(* Logix 5000 project; controller AMANA_DC_PLANT_01 vendor 1 type 14 code 164 rev 31.12; software revision 31.02; part 3 of 9 *)
(* tags used below, declared in another part *)
   Break1_Hour : DINT;
   Break1_Hour_String : STRING_4;
   Break1_Length : DINT;
   Break1_Min : DINT;
   Break1_Min_String : STRING_4;
   Break2_Hour : DINT;
   Break2_Hour_String : STRING_4;
   Break2_Length : DINT;
   Break2_Min : DINT;
   Break2_Min_String : STRING_4;
   End_Hour : DINT;
   End_Hour_String : STRING_4;
   End_Min : DINT;
   End_Min_String : STRING_4;
   Lunch_Hour : DINT;
   Lunch_Hour_String : STRING_4;
   Lunch_Length : DINT;
   Lunch_Min : DINT;
   Lunch_Min_String : STRING_4;
   PreviousCount : DINT;
   Shift_Reset : BOOL;
   Start_Hour : DINT;
   Start_Hour_String : STRING_4;
   Start_Min : DINT;
   Start_Min_String : STRING_4;
   theoreticalUnitsReal : REAL;
   ay : REAL;
   fifi_unload : DINT;
   LN00_Schedule : UDT_Current_Status;
   LN00_ScheduleUnits_Produced_from_line : DINT;
   LN00_to_DC1_Main_Messages_0 : DINT[40];
   LN00_Toggle_CountSource : BOOL;
   LN00_Weekly_Schedule : UDT_Weekly_Schedule;
   null : STRING;
   Previous_Shift_Count : DINT;
   scc : CONTROL;   // Shift Count History
   Shift_count_history : DINT[62];
   Shift_reset_timer : TIMER;
   THEORETICAL_TEST : BOOL;
(* LN00, continued *)

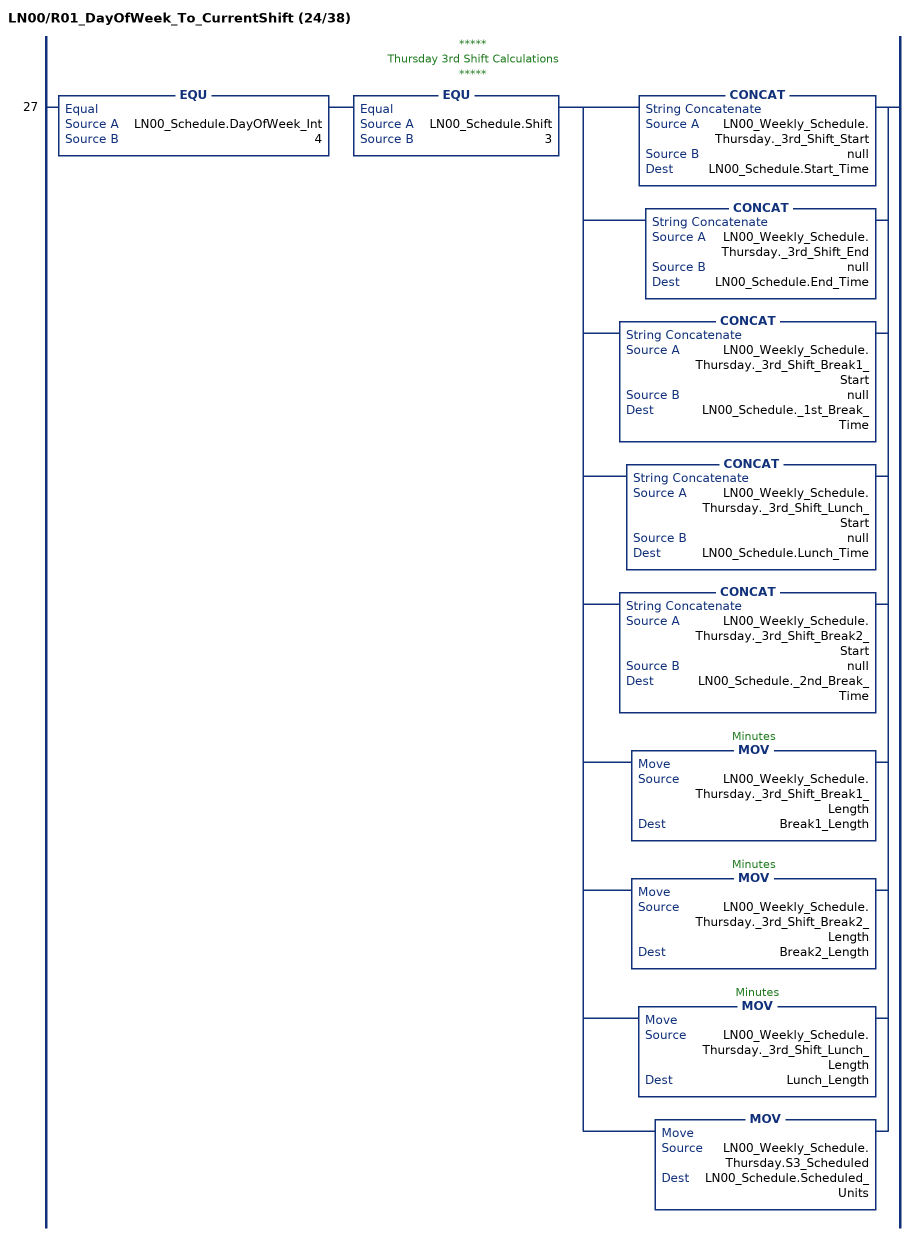
   [picture p24: LN00/R01_DayOfWeek_To_CurrentShift rungs 27-27]
   // *****
   // Thursday 3rd Shift Calculations
   // *****
   27: EQU(LN00_Schedule.DayOfWeek_Int,4)EQU(LN00_Schedule.Shift,3)[CONCAT(LN00_Weekly_Schedule.Thursday._3rd_Shift_Start,null,LN00_Schedule.Start_Time) ,CONCAT(LN00_Weekly_Schedule.Thursday._3rd_Shift_End,null,LN00_Schedule.End_Time) ,CONCAT(LN00_Weekly_Schedule.Thursday._3rd_Shift_Break1_Start,null,LN00_Schedule._1st_Break_Time) ,CONCAT(LN00_Weekly_Schedule.Thursday._3rd_Shift_Lunch_Start,null,LN00_Schedule.Lunch_Time) ,CONCAT(LN00_Weekly_Schedule.Thursday._3rd_Shift_Break2_Start,null,LN00_Schedule._2nd_Break_Time) ,MOV(LN00_Weekly_Schedule.Thursday._3rd_Shift_Break1_Length,Break1_Length) ,MOV(LN00_Weekly_Schedule.Thursday._3rd_Shift_Break2_Length,Break2_Length) ,MOV(LN00_Weekly_Schedule.Thursday._3rd_Shift_Lunch_Length,Lunch_Length) ,MOV(LN00_Weekly_Schedule.Thursday.S3_Scheduled,LN00_Schedule.Scheduled_Units) ];
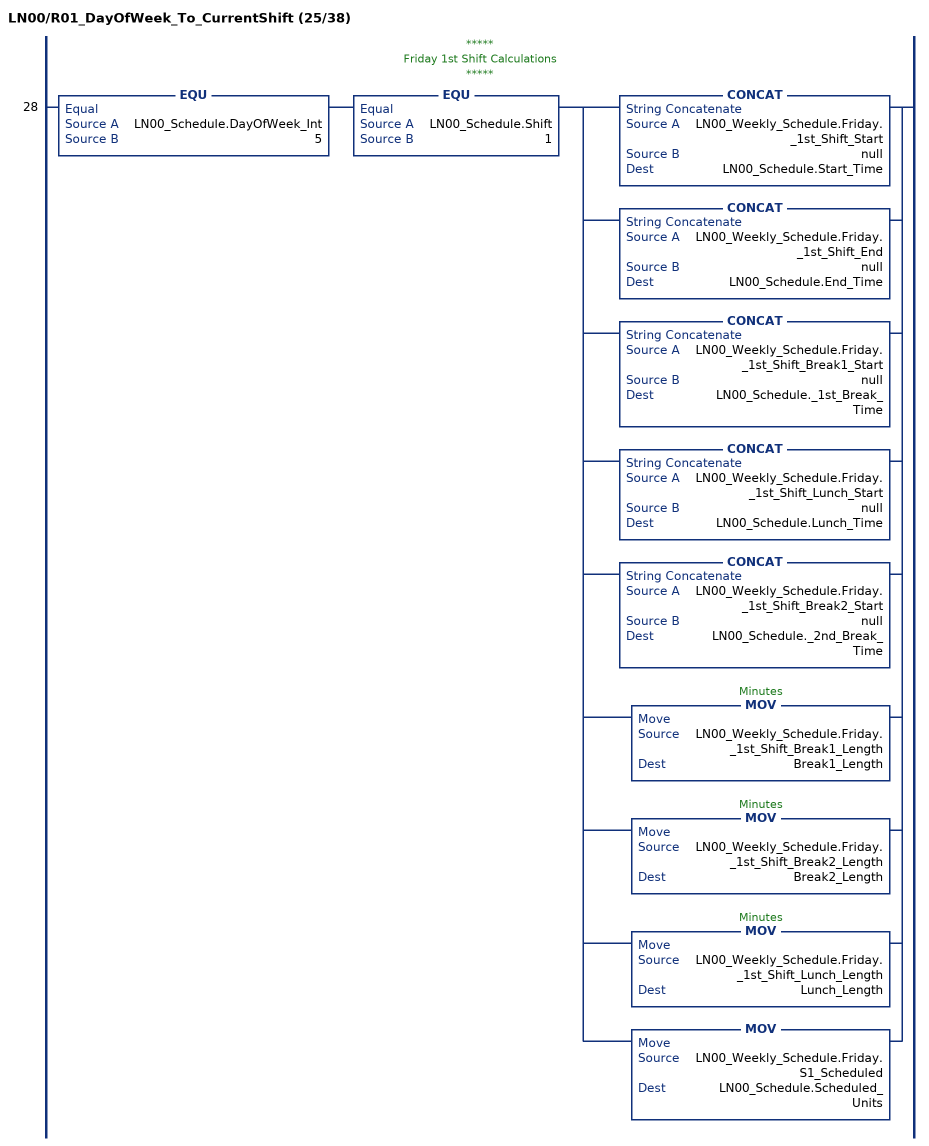
   // *****
   // Friday 1st Shift Calculations
   // *****
   28: EQU(LN00_Schedule.DayOfWeek_Int,5)EQU(LN00_Schedule.Shift,1)[CONCAT(LN00_Weekly_Schedule.Friday._1st_Shift_Start,null,LN00_Schedule.Start_Time) ,CONCAT(LN00_Weekly_Schedule.Friday._1st_Shift_End,null,LN00_Schedule.End_Time) ,CONCAT(LN00_Weekly_Schedule.Friday._1st_Shift_Break1_Start,null,LN00_Schedule._1st_Break_Time) ,CONCAT(LN00_Weekly_Schedule.Friday._1st_Shift_Lunch_Start,null,LN00_Schedule.Lunch_Time) ,CONCAT(LN00_Weekly_Schedule.Friday._1st_Shift_Break2_Start,null,LN00_Schedule._2nd_Break_Time) ,MOV(LN00_Weekly_Schedule.Friday._1st_Shift_Break1_Length,Break1_Length) ,MOV(LN00_Weekly_Schedule.Friday._1st_Shift_Break2_Length,Break2_Length) ,MOV(LN00_Weekly_Schedule.Friday._1st_Shift_Lunch_Length,Lunch_Length) ,MOV(LN00_Weekly_Schedule.Friday.S1_Scheduled,LN00_Schedule.Scheduled_Units) ];
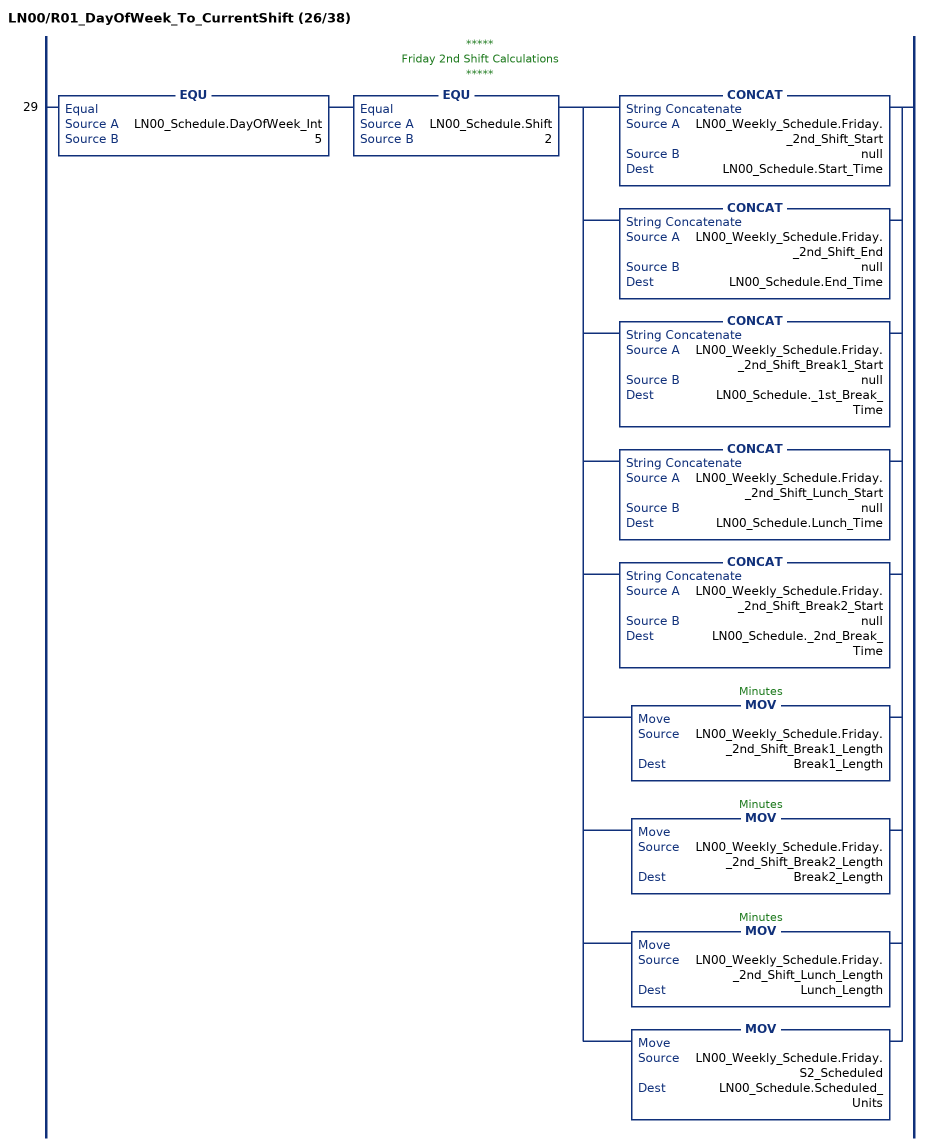
   // *****
   // Friday 2nd Shift Calculations
   // *****
   29: EQU(LN00_Schedule.DayOfWeek_Int,5)EQU(LN00_Schedule.Shift,2)[CONCAT(LN00_Weekly_Schedule.Friday._2nd_Shift_Start,null,LN00_Schedule.Start_Time) ,CONCAT(LN00_Weekly_Schedule.Friday._2nd_Shift_End,null,LN00_Schedule.End_Time) ,CONCAT(LN00_Weekly_Schedule.Friday._2nd_Shift_Break1_Start,null,LN00_Schedule._1st_Break_Time) ,CONCAT(LN00_Weekly_Schedule.Friday._2nd_Shift_Lunch_Start,null,LN00_Schedule.Lunch_Time) ,CONCAT(LN00_Weekly_Schedule.Friday._2nd_Shift_Break2_Start,null,LN00_Schedule._2nd_Break_Time) ,MOV(LN00_Weekly_Schedule.Friday._2nd_Shift_Break1_Length,Break1_Length) ,MOV(LN00_Weekly_Schedule.Friday._2nd_Shift_Break2_Length,Break2_Length) ,MOV(LN00_Weekly_Schedule.Friday._2nd_Shift_Lunch_Length,Lunch_Length) ,MOV(LN00_Weekly_Schedule.Friday.S2_Scheduled,LN00_Schedule.Scheduled_Units) ];
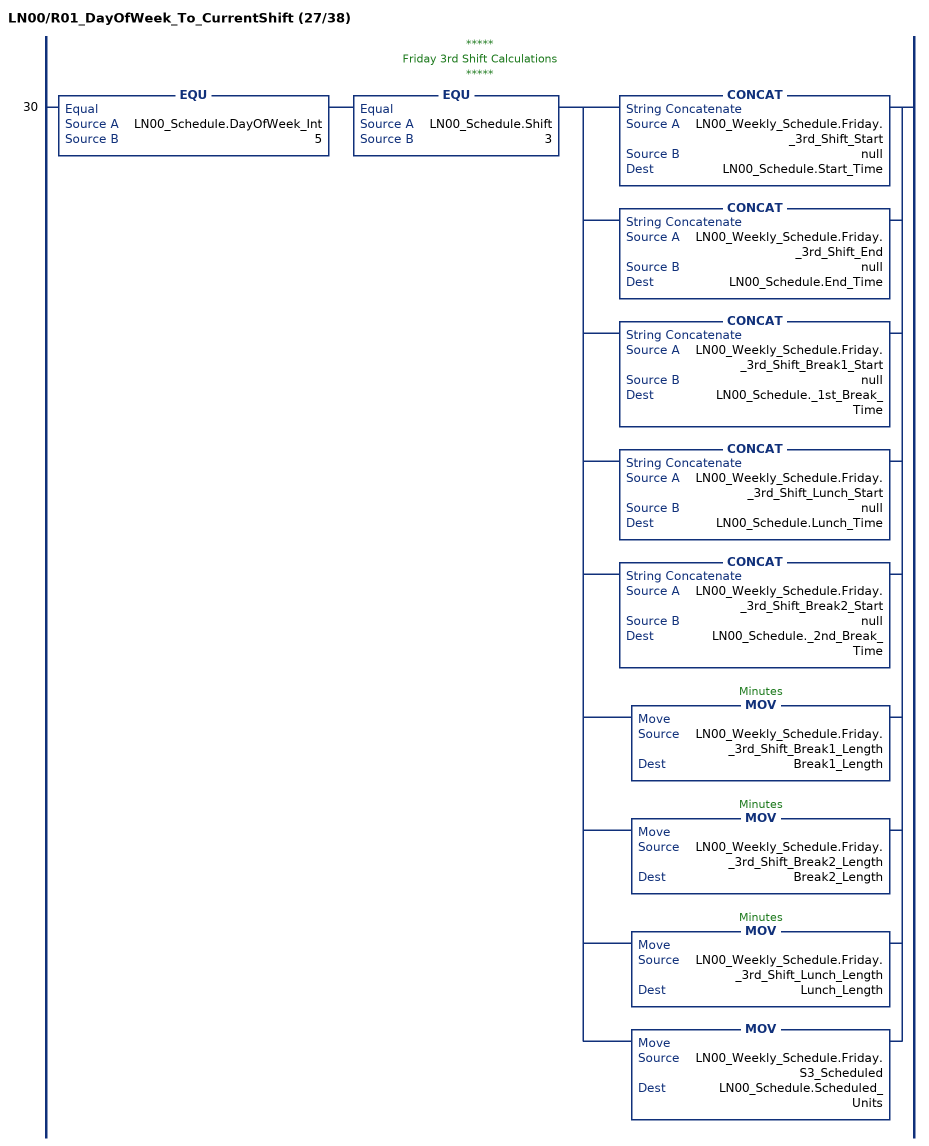
   // *****
   // Friday 3rd Shift Calculations
   // *****
   30: EQU(LN00_Schedule.DayOfWeek_Int,5)EQU(LN00_Schedule.Shift,3)[CONCAT(LN00_Weekly_Schedule.Friday._3rd_Shift_Start,null,LN00_Schedule.Start_Time) ,CONCAT(LN00_Weekly_Schedule.Friday._3rd_Shift_End,null,LN00_Schedule.End_Time) ,CONCAT(LN00_Weekly_Schedule.Friday._3rd_Shift_Break1_Start,null,LN00_Schedule._1st_Break_Time) ,CONCAT(LN00_Weekly_Schedule.Friday._3rd_Shift_Lunch_Start,null,LN00_Schedule.Lunch_Time) ,CONCAT(LN00_Weekly_Schedule.Friday._3rd_Shift_Break2_Start,null,LN00_Schedule._2nd_Break_Time) ,MOV(LN00_Weekly_Schedule.Friday._3rd_Shift_Break1_Length,Break1_Length) ,MOV(LN00_Weekly_Schedule.Friday._3rd_Shift_Break2_Length,Break2_Length) ,MOV(LN00_Weekly_Schedule.Friday._3rd_Shift_Lunch_Length,Lunch_Length) ,MOV(LN00_Weekly_Schedule.Friday.S3_Scheduled,LN00_Schedule.Scheduled_Units) ];
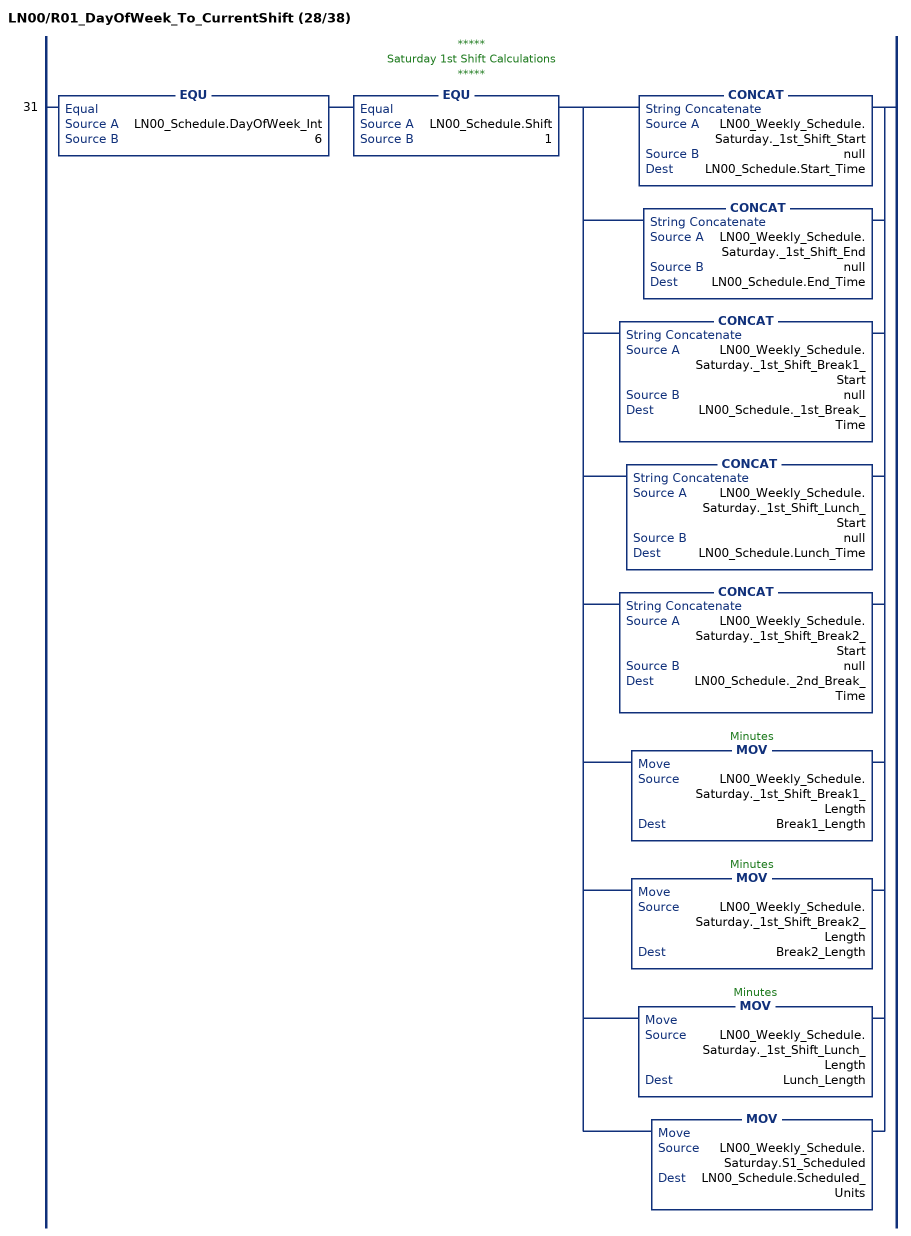
   // *****
   // Saturday 1st Shift Calculations
   // *****
   31: EQU(LN00_Schedule.DayOfWeek_Int,6)EQU(LN00_Schedule.Shift,1)[CONCAT(LN00_Weekly_Schedule.Saturday._1st_Shift_Start,null,LN00_Schedule.Start_Time) ,CONCAT(LN00_Weekly_Schedule.Saturday._1st_Shift_End,null,LN00_Schedule.End_Time) ,CONCAT(LN00_Weekly_Schedule.Saturday._1st_Shift_Break1_Start,null,LN00_Schedule._1st_Break_Time) ,CONCAT(LN00_Weekly_Schedule.Saturday._1st_Shift_Lunch_Start,null,LN00_Schedule.Lunch_Time) ,CONCAT(LN00_Weekly_Schedule.Saturday._1st_Shift_Break2_Start,null,LN00_Schedule._2nd_Break_Time) ,MOV(LN00_Weekly_Schedule.Saturday._1st_Shift_Break1_Length,Break1_Length) ,MOV(LN00_Weekly_Schedule.Saturday._1st_Shift_Break2_Length,Break2_Length) ,MOV(LN00_Weekly_Schedule.Saturday._1st_Shift_Lunch_Length,Lunch_Length) ,MOV(LN00_Weekly_Schedule.Saturday.S1_Scheduled,LN00_Schedule.Scheduled_Units) ];
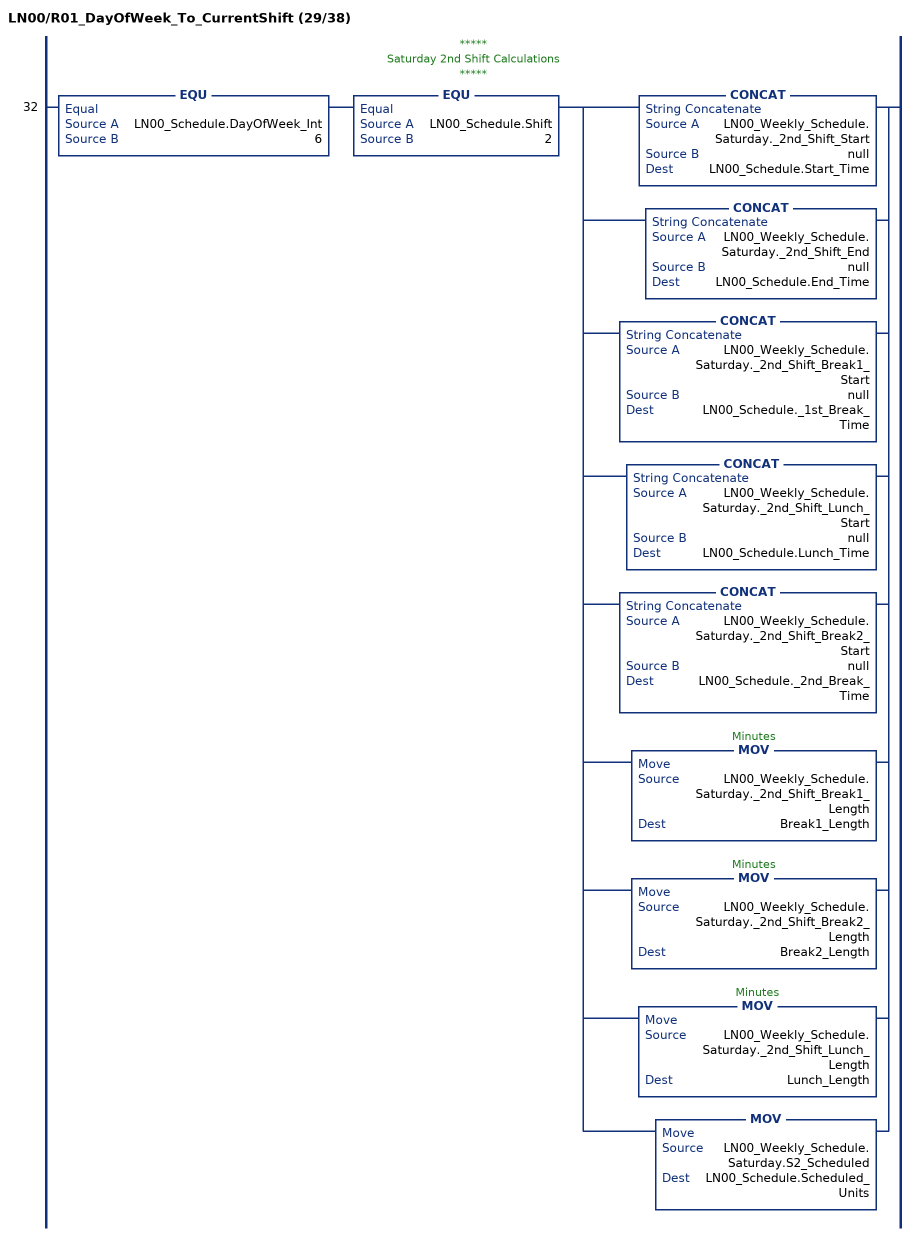
   // *****
   // Saturday 2nd Shift Calculations
   // *****
   32: EQU(LN00_Schedule.DayOfWeek_Int,6)EQU(LN00_Schedule.Shift,2)[CONCAT(LN00_Weekly_Schedule.Saturday._2nd_Shift_Start,null,LN00_Schedule.Start_Time) ,CONCAT(LN00_Weekly_Schedule.Saturday._2nd_Shift_End,null,LN00_Schedule.End_Time) ,CONCAT(LN00_Weekly_Schedule.Saturday._2nd_Shift_Break1_Start,null,LN00_Schedule._1st_Break_Time) ,CONCAT(LN00_Weekly_Schedule.Saturday._2nd_Shift_Lunch_Start,null,LN00_Schedule.Lunch_Time) ,CONCAT(LN00_Weekly_Schedule.Saturday._2nd_Shift_Break2_Start,null,LN00_Schedule._2nd_Break_Time) ,MOV(LN00_Weekly_Schedule.Saturday._2nd_Shift_Break1_Length,Break1_Length) ,MOV(LN00_Weekly_Schedule.Saturday._2nd_Shift_Break2_Length,Break2_Length) ,MOV(LN00_Weekly_Schedule.Saturday._2nd_Shift_Lunch_Length,Lunch_Length) ,MOV(LN00_Weekly_Schedule.Saturday.S2_Scheduled,LN00_Schedule.Scheduled_Units) ];
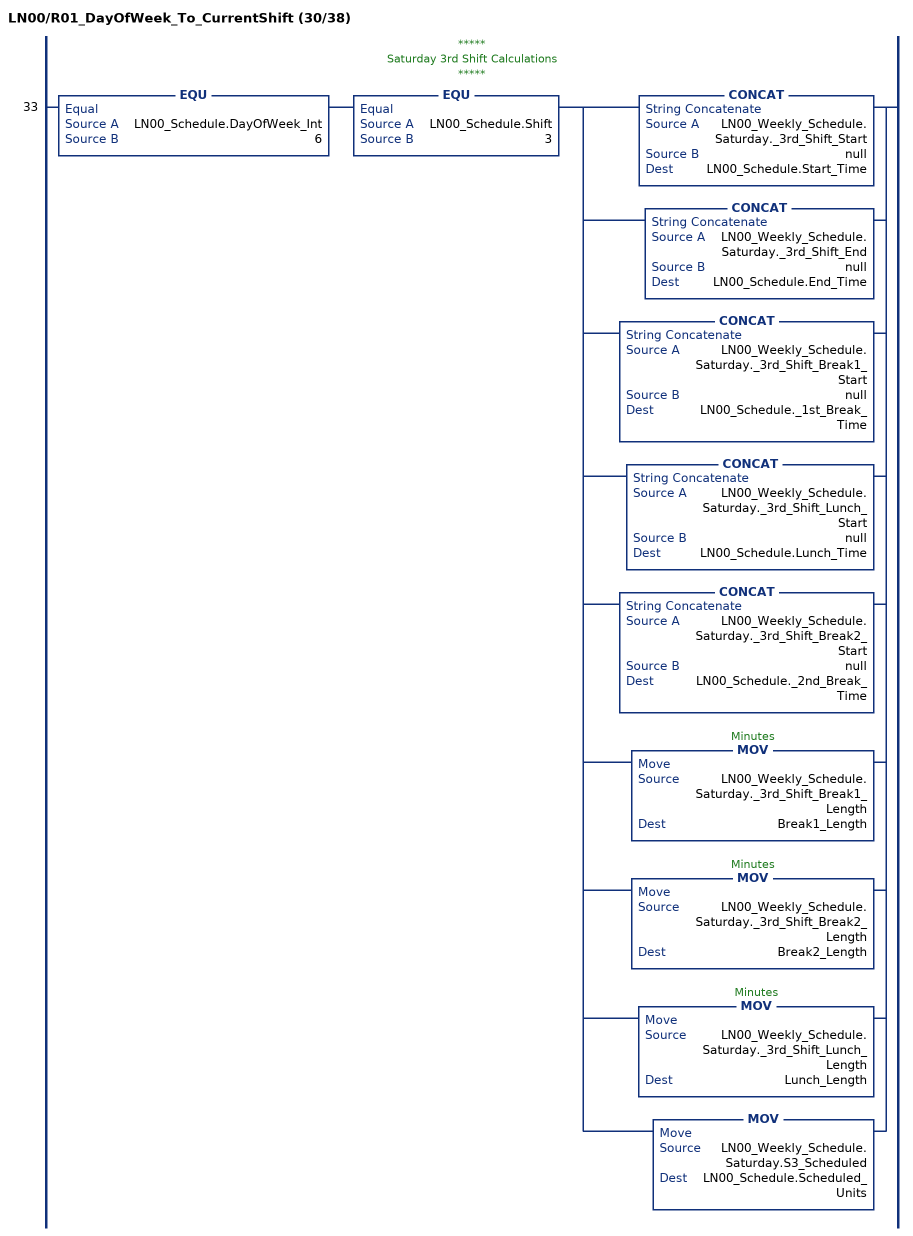
   // *****
   // Saturday 3rd Shift Calculations
   // *****
   33: EQU(LN00_Schedule.DayOfWeek_Int,6)EQU(LN00_Schedule.Shift,3)[CONCAT(LN00_Weekly_Schedule.Saturday._3rd_Shift_Start,null,LN00_Schedule.Start_Time) ,CONCAT(LN00_Weekly_Schedule.Saturday._3rd_Shift_End,null,LN00_Schedule.End_Time) ,CONCAT(LN00_Weekly_Schedule.Saturday._3rd_Shift_Break1_Start,null,LN00_Schedule._1st_Break_Time) ,CONCAT(LN00_Weekly_Schedule.Saturday._3rd_Shift_Lunch_Start,null,LN00_Schedule.Lunch_Time) ,CONCAT(LN00_Weekly_Schedule.Saturday._3rd_Shift_Break2_Start,null,LN00_Schedule._2nd_Break_Time) ,MOV(LN00_Weekly_Schedule.Saturday._3rd_Shift_Break1_Length,Break1_Length) ,MOV(LN00_Weekly_Schedule.Saturday._3rd_Shift_Break2_Length,Break2_Length) ,MOV(LN00_Weekly_Schedule.Saturday._3rd_Shift_Lunch_Length,Lunch_Length) ,MOV(LN00_Weekly_Schedule.Saturday.S3_Scheduled,LN00_Schedule.Scheduled_Units) ];
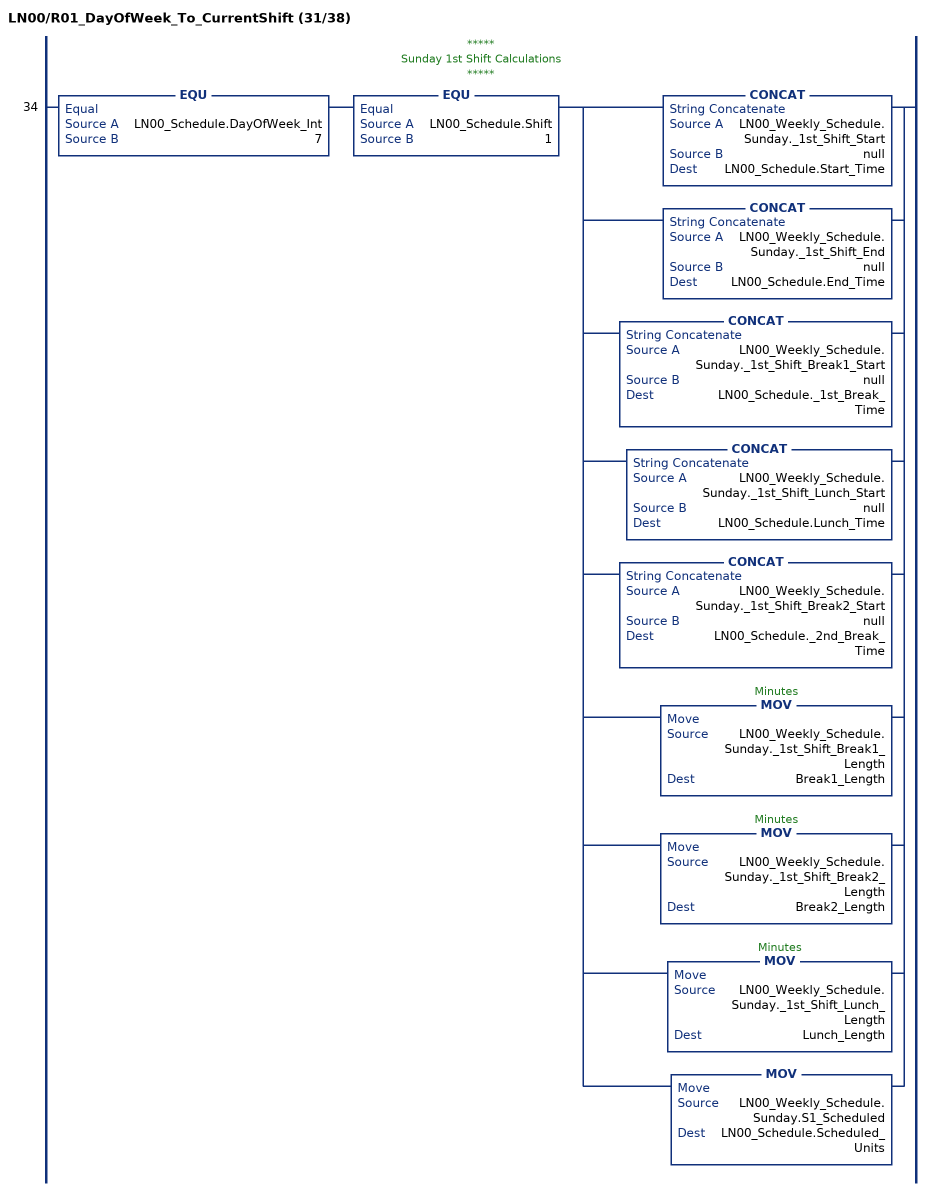
   // *****
   // Sunday 1st Shift Calculations
   // *****
   34: EQU(LN00_Schedule.DayOfWeek_Int,7)EQU(LN00_Schedule.Shift,1)[CONCAT(LN00_Weekly_Schedule.Sunday._1st_Shift_Start,null,LN00_Schedule.Start_Time) ,CONCAT(LN00_Weekly_Schedule.Sunday._1st_Shift_End,null,LN00_Schedule.End_Time) ,CONCAT(LN00_Weekly_Schedule.Sunday._1st_Shift_Break1_Start,null,LN00_Schedule._1st_Break_Time) ,CONCAT(LN00_Weekly_Schedule.Sunday._1st_Shift_Lunch_Start,null,LN00_Schedule.Lunch_Time) ,CONCAT(LN00_Weekly_Schedule.Sunday._1st_Shift_Break2_Start,null,LN00_Schedule._2nd_Break_Time) ,MOV(LN00_Weekly_Schedule.Sunday._1st_Shift_Break1_Length,Break1_Length) ,MOV(LN00_Weekly_Schedule.Sunday._1st_Shift_Break2_Length,Break2_Length) ,MOV(LN00_Weekly_Schedule.Sunday._1st_Shift_Lunch_Length,Lunch_Length) ,MOV(LN00_Weekly_Schedule.Sunday.S1_Scheduled,LN00_Schedule.Scheduled_Units) ];
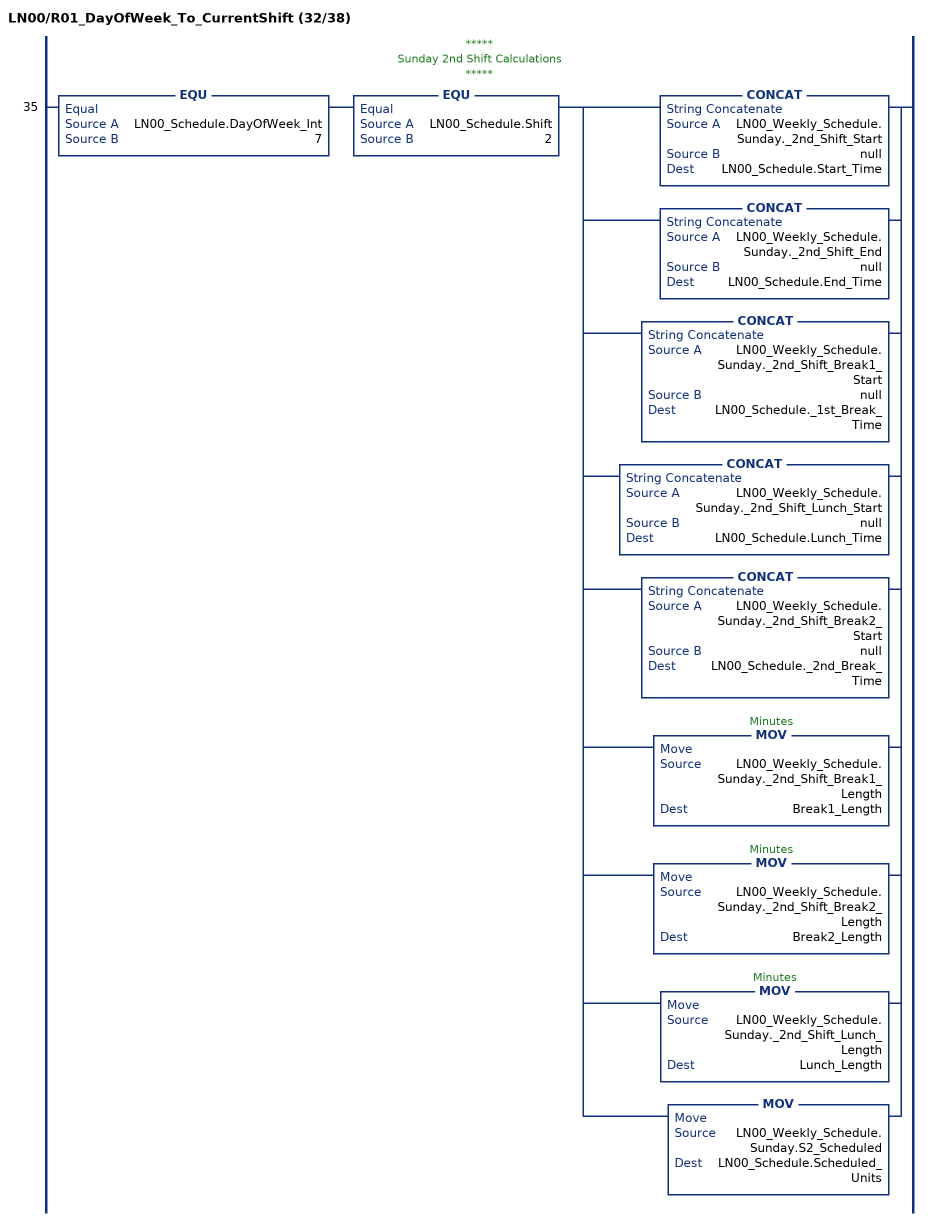
   // *****
   // Sunday 2nd Shift Calculations
   // *****
   35: EQU(LN00_Schedule.DayOfWeek_Int,7)EQU(LN00_Schedule.Shift,2)[CONCAT(LN00_Weekly_Schedule.Sunday._2nd_Shift_Start,null,LN00_Schedule.Start_Time) ,CONCAT(LN00_Weekly_Schedule.Sunday._2nd_Shift_End,null,LN00_Schedule.End_Time) ,CONCAT(LN00_Weekly_Schedule.Sunday._2nd_Shift_Break1_Start,null,LN00_Schedule._1st_Break_Time) ,CONCAT(LN00_Weekly_Schedule.Sunday._2nd_Shift_Lunch_Start,null,LN00_Schedule.Lunch_Time) ,CONCAT(LN00_Weekly_Schedule.Sunday._2nd_Shift_Break2_Start,null,LN00_Schedule._2nd_Break_Time) ,MOV(LN00_Weekly_Schedule.Sunday._2nd_Shift_Break1_Length,Break1_Length) ,MOV(LN00_Weekly_Schedule.Sunday._2nd_Shift_Break2_Length,Break2_Length) ,MOV(LN00_Weekly_Schedule.Sunday._2nd_Shift_Lunch_Length,Lunch_Length) ,MOV(LN00_Weekly_Schedule.Sunday.S2_Scheduled,LN00_Schedule.Scheduled_Units) ];
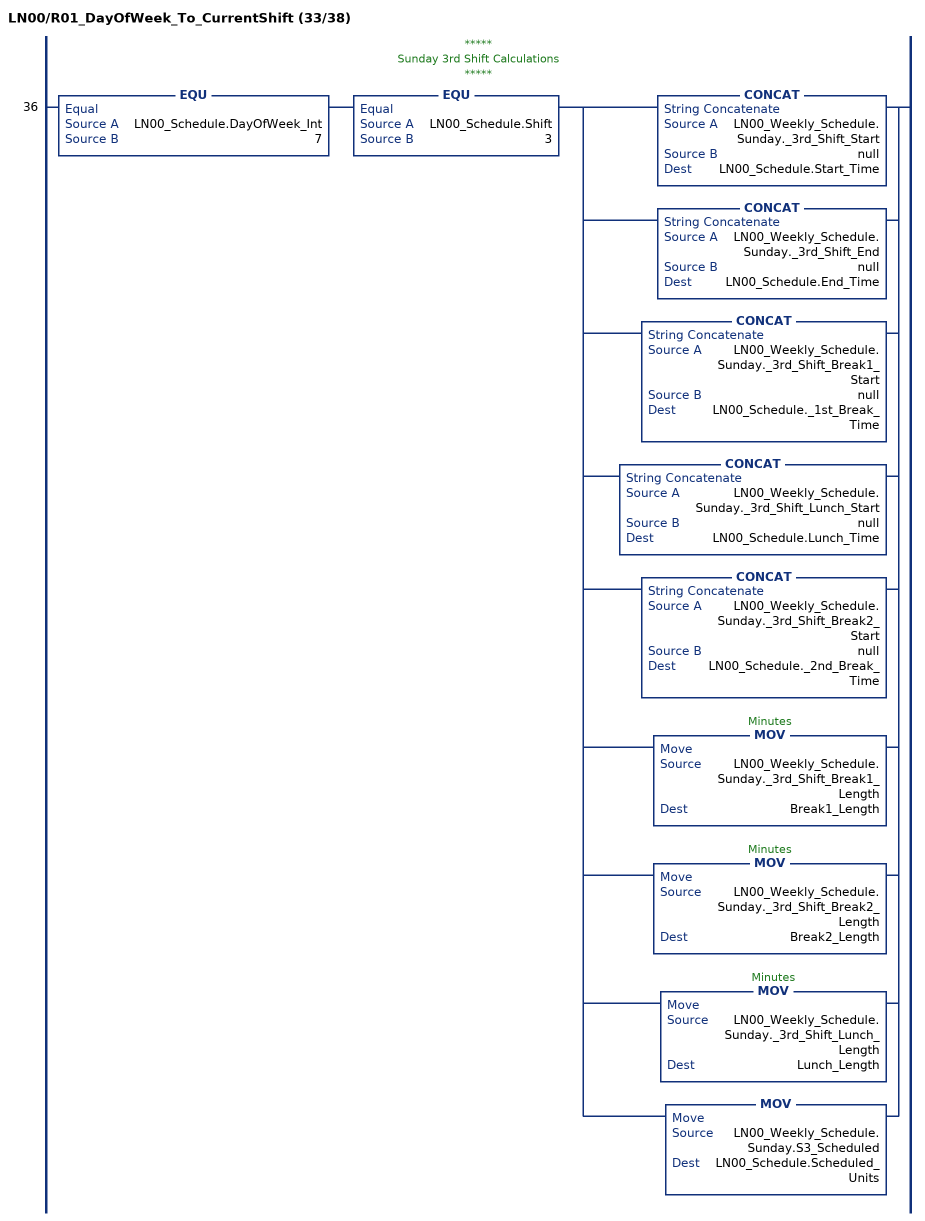
   // *****
   // Sunday 3rd Shift Calculations
   // *****
   36: EQU(LN00_Schedule.DayOfWeek_Int,7)EQU(LN00_Schedule.Shift,3)[CONCAT(LN00_Weekly_Schedule.Sunday._3rd_Shift_Start,null,LN00_Schedule.Start_Time) ,CONCAT(LN00_Weekly_Schedule.Sunday._3rd_Shift_End,null,LN00_Schedule.End_Time) ,CONCAT(LN00_Weekly_Schedule.Sunday._3rd_Shift_Break1_Start,null,LN00_Schedule._1st_Break_Time) ,CONCAT(LN00_Weekly_Schedule.Sunday._3rd_Shift_Lunch_Start,null,LN00_Schedule.Lunch_Time) ,CONCAT(LN00_Weekly_Schedule.Sunday._3rd_Shift_Break2_Start,null,LN00_Schedule._2nd_Break_Time) ,MOV(LN00_Weekly_Schedule.Sunday._3rd_Shift_Break1_Length,Break1_Length) ,MOV(LN00_Weekly_Schedule.Sunday._3rd_Shift_Break2_Length,Break2_Length) ,MOV(LN00_Weekly_Schedule.Sunday._3rd_Shift_Lunch_Length,Lunch_Length) ,MOV(LN00_Weekly_Schedule.Sunday.S3_Scheduled,LN00_Schedule.Scheduled_Units) ];
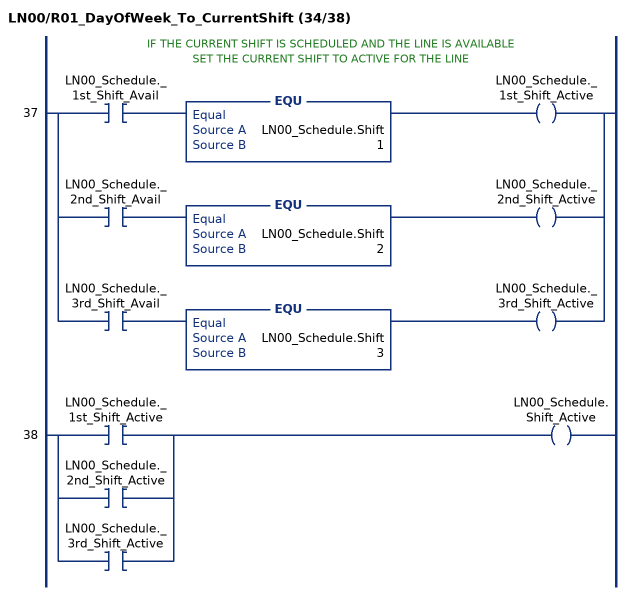
   // IF THE CURRENT SHIFT IS SCHEDULED AND THE LINE IS AVAILABLE
   // SET THE CURRENT SHIFT TO ACTIVE FOR THE LINE
   37: [XIC(LN00_Schedule._1st_Shift_Avail) EQU(LN00_Schedule.Shift,1) OTE(LN00_Schedule._1st_Shift_Active) ,XIC(LN00_Schedule._2nd_Shift_Avail) EQU(LN00_Schedule.Shift,2) OTE(LN00_Schedule._2nd_Shift_Active) ,XIC(LN00_Schedule._3rd_Shift_Avail) EQU(LN00_Schedule.Shift,3) OTE(LN00_Schedule._3rd_Shift_Active) ];
   38: [XIC(LN00_Schedule._1st_Shift_Active) ,XIC(LN00_Schedule._2nd_Shift_Active) ,XIC(LN00_Schedule._3rd_Shift_Active) ]OTE(LN00_Schedule.Shift_Active);
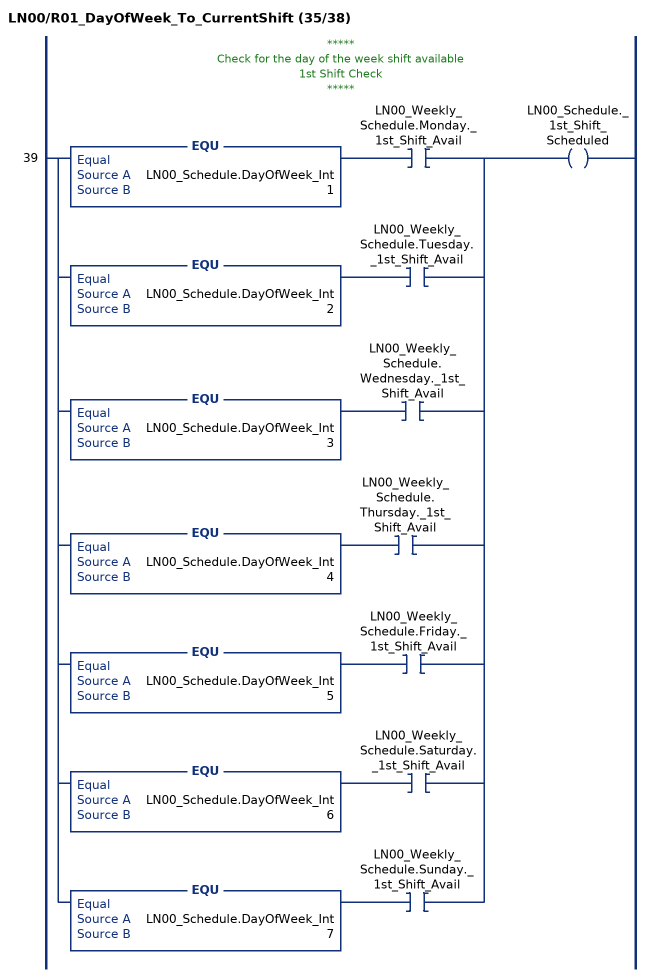
   // *****
   // Check for the day of the week shift available
   // 1st Shift Check
   // *****
   39: [EQU(LN00_Schedule.DayOfWeek_Int,1) XIC(LN00_Weekly_Schedule.Monday._1st_Shift_Avail) ,EQU(LN00_Schedule.DayOfWeek_Int,2) XIC(LN00_Weekly_Schedule.Tuesday._1st_Shift_Avail) ,EQU(LN00_Schedule.DayOfWeek_Int,3) XIC(LN00_Weekly_Schedule.Wednesday._1st_Shift_Avail) ,EQU(LN00_Schedule.DayOfWeek_Int,4) XIC(LN00_Weekly_Schedule.Thursday._1st_Shift_Avail) ,EQU(LN00_Schedule.DayOfWeek_Int,5) XIC(LN00_Weekly_Schedule.Friday._1st_Shift_Avail) ,EQU(LN00_Schedule.DayOfWeek_Int,6) XIC(LN00_Weekly_Schedule.Saturday._1st_Shift_Avail) ,EQU(LN00_Schedule.DayOfWeek_Int,7) XIC(LN00_Weekly_Schedule.Sunday._1st_Shift_Avail) ]OTE(LN00_Schedule._1st_Shift_Scheduled);
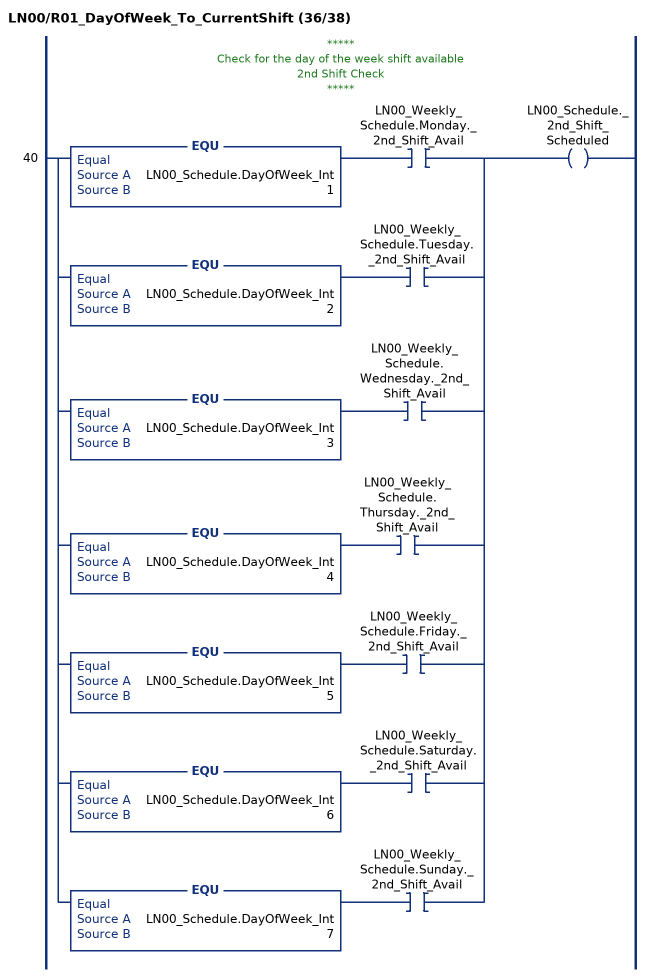
   // *****
   // Check for the day of the week shift available
   // 2nd Shift Check
   // *****
   40: [EQU(LN00_Schedule.DayOfWeek_Int,1) XIC(LN00_Weekly_Schedule.Monday._2nd_Shift_Avail) ,EQU(LN00_Schedule.DayOfWeek_Int,2) XIC(LN00_Weekly_Schedule.Tuesday._2nd_Shift_Avail) ,EQU(LN00_Schedule.DayOfWeek_Int,3) XIC(LN00_Weekly_Schedule.Wednesday._2nd_Shift_Avail) ,EQU(LN00_Schedule.DayOfWeek_Int,4) XIC(LN00_Weekly_Schedule.Thursday._2nd_Shift_Avail) ,EQU(LN00_Schedule.DayOfWeek_Int,5) XIC(LN00_Weekly_Schedule.Friday._2nd_Shift_Avail) ,EQU(LN00_Schedule.DayOfWeek_Int,6) XIC(LN00_Weekly_Schedule.Saturday._2nd_Shift_Avail) ,EQU(LN00_Schedule.DayOfWeek_Int,7) XIC(LN00_Weekly_Schedule.Sunday._2nd_Shift_Avail) ]OTE(LN00_Schedule._2nd_Shift_Scheduled);
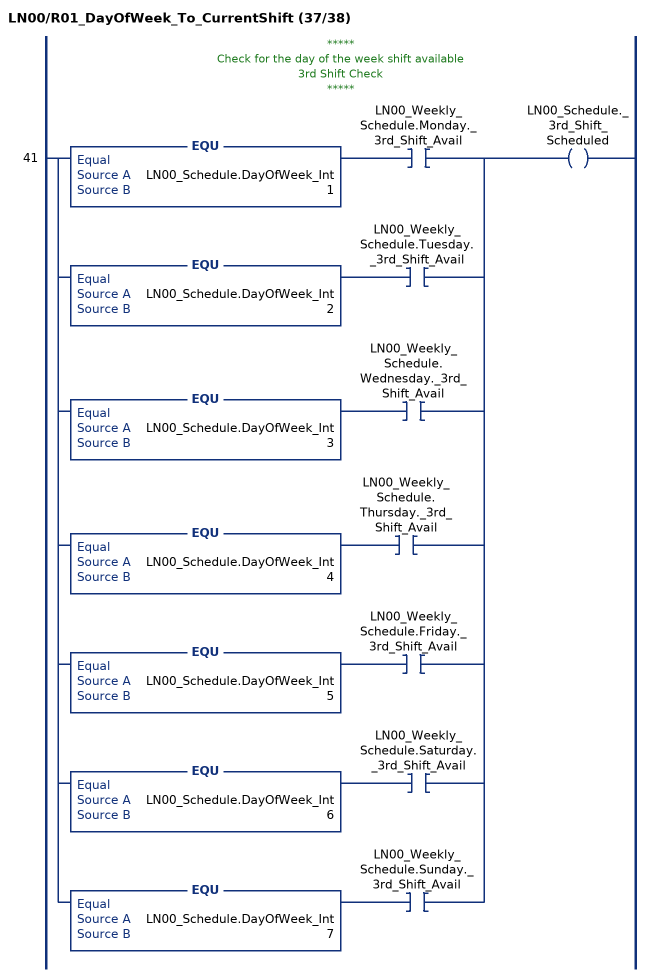
   // *****
   // Check for the day of the week shift available
   // 3rd Shift Check
   // *****
   41: [EQU(LN00_Schedule.DayOfWeek_Int,1) XIC(LN00_Weekly_Schedule.Monday._3rd_Shift_Avail) ,EQU(LN00_Schedule.DayOfWeek_Int,2) XIC(LN00_Weekly_Schedule.Tuesday._3rd_Shift_Avail) ,EQU(LN00_Schedule.DayOfWeek_Int,3) XIC(LN00_Weekly_Schedule.Wednesday._3rd_Shift_Avail) ,EQU(LN00_Schedule.DayOfWeek_Int,4) XIC(LN00_Weekly_Schedule.Thursday._3rd_Shift_Avail) ,EQU(LN00_Schedule.DayOfWeek_Int,5) XIC(LN00_Weekly_Schedule.Friday._3rd_Shift_Avail) ,EQU(LN00_Schedule.DayOfWeek_Int,6) XIC(LN00_Weekly_Schedule.Saturday._3rd_Shift_Avail) ,EQU(LN00_Schedule.DayOfWeek_Int,7) XIC(LN00_Weekly_Schedule.Sunday._3rd_Shift_Avail) ]OTE(LN00_Schedule._3rd_Shift_Scheduled);
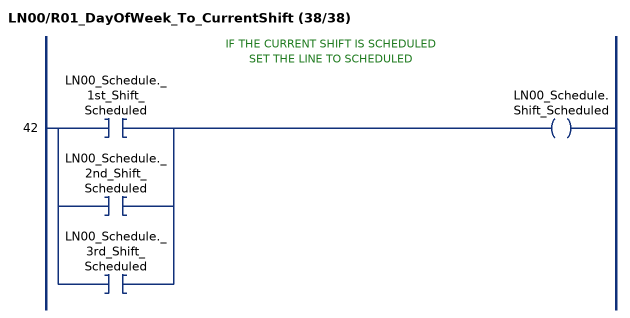
   // IF THE CURRENT SHIFT IS SCHEDULED
   // SET THE LINE TO SCHEDULED
   42: [XIC(LN00_Schedule._1st_Shift_Scheduled) ,XIC(LN00_Schedule._2nd_Shift_Scheduled) ,XIC(LN00_Schedule._3rd_Shift_Scheduled) ]OTE(LN00_Schedule.Shift_Scheduled);
END_ROUTINE

ROUTINE R02_CurrentShift_Calcs   (* ladder *)
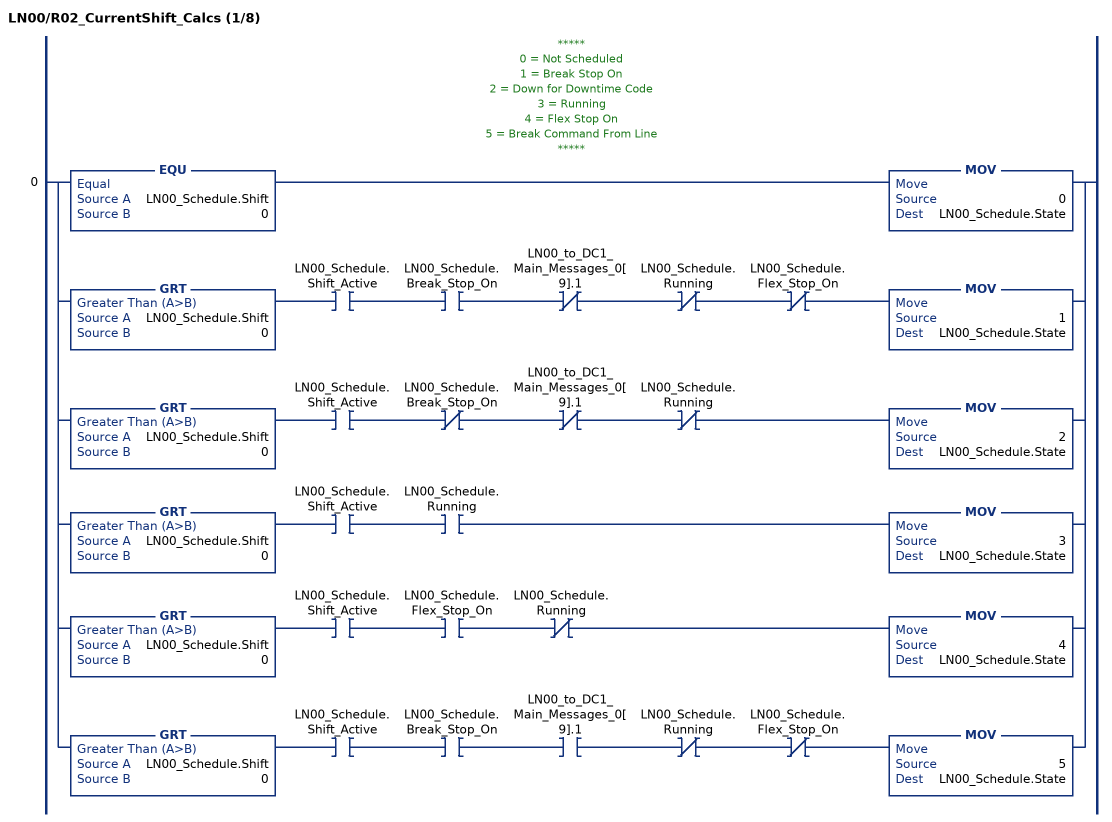
   // *****
   // 0 = Not Scheduled
   // 1 = Break Stop On
   // 2 = Down for Downtime Code
   // 3 = Running
   // 4 = Flex Stop On
   // 5 = Break Command From Line
   // *****
   0: [EQU(LN00_Schedule.Shift,0) MOV(0,LN00_Schedule.State) ,GRT(LN00_Schedule.Shift,0) XIC(LN00_Schedule.Shift_Active) XIC(LN00_Schedule.Break_Stop_On) XIO(LN00_to_DC1_Main_Messages_0[9].1) XIO(LN00_Schedule.Running) XIO(LN00_Schedule.Flex_Stop_On) MOV(1,LN00_Schedule.State) ,GRT(LN00_Schedule.Shift,0) XIC(LN00_Schedule.Shift_Active) XIO(LN00_Schedule.Break_Stop_On) XIO(LN00_to_DC1_Main_Messages_0[9].1) XIO(LN00_Schedule.Running) MOV(2,LN00_Schedule.State) ,GRT(LN00_Schedule.Shift,0) XIC(LN00_Schedule.Shift_Active) XIC(LN00_Schedule.Running) MOV(3,LN00_Schedule.State) ,GRT(LN00_Schedule.Shift,0) XIC(LN00_Schedule.Shift_Active) XIC(LN00_Schedule.Flex_Stop_On) XIO(LN00_Schedule.Running) MOV(4,LN00_Schedule.State) ,GRT(LN00_Schedule.Shift,0) XIC(LN00_Schedule.Shift_Active) XIC(LN00_Schedule.Break_Stop_On) XIC(LN00_to_DC1_Main_Messages_0[9].1) XIO(LN00_Schedule.Running) XIO(LN00_Schedule.Flex_Stop_On) MOV(5,LN00_Schedule.State) ];
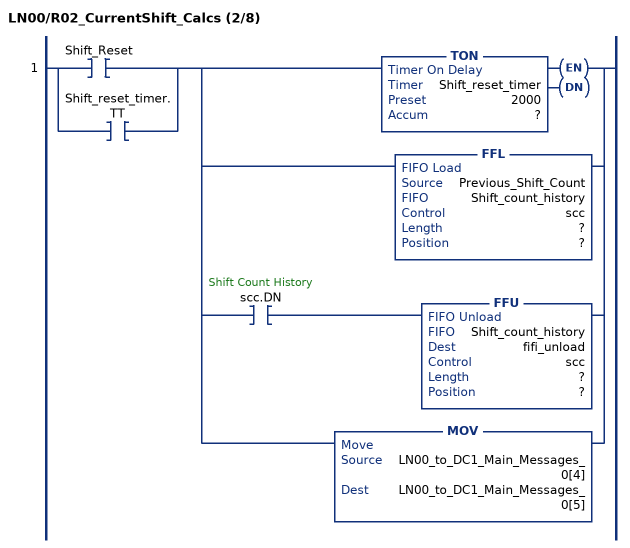
   1: [XIC(Shift_Reset) ,XIC(Shift_reset_timer.TT) ][TON(Shift_reset_timer,?,?) ,FFL(Previous_Shift_Count,Shift_count_history,scc,?,?) ,XIC(scc.DN) FFU(Shift_count_history,fifi_unload,scc,?,?) ,MOV(LN00_to_DC1_Main_Messages_0[4],LN00_to_DC1_Main_Messages_0[5]) ];
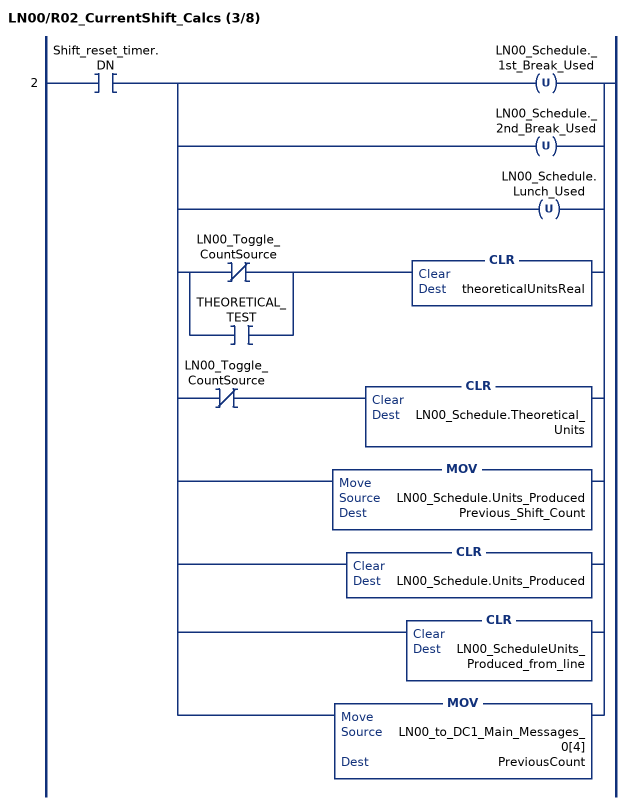
   2: XIC(Shift_reset_timer.DN)[OTU(LN00_Schedule._1st_Break_Used) ,OTU(LN00_Schedule._2nd_Break_Used) ,OTU(LN00_Schedule.Lunch_Used) ,[XIO(LN00_Toggle_CountSource) ,XIC(THEORETICAL_TEST) ] CLR(theoreticalUnitsReal) ,XIO(LN00_Toggle_CountSource) CLR(LN00_Schedule.Theoretical_Units) ,MOV(LN00_Schedule.Units_Produced,Previous_Shift_Count) ,CLR(LN00_Schedule.Units_Produced) ,CLR(LN00_ScheduleUnits_Produced_from_line) ,MOV(LN00_to_DC1_Main_Messages_0[4],PreviousCount) ];
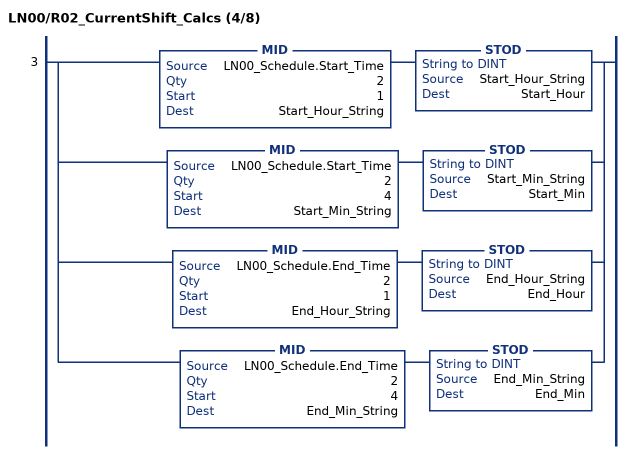
   3: [MID(LN00_Schedule.Start_Time,2,1,Start_Hour_String) STOD(Start_Hour_String,Start_Hour) ,MID(LN00_Schedule.Start_Time,2,4,Start_Min_String) STOD(Start_Min_String,Start_Min) ,MID(LN00_Schedule.End_Time,2,1,End_Hour_String) STOD(End_Hour_String,End_Hour) ,MID(LN00_Schedule.End_Time,2,4,End_Min_String) STOD(End_Min_String,End_Min) ];
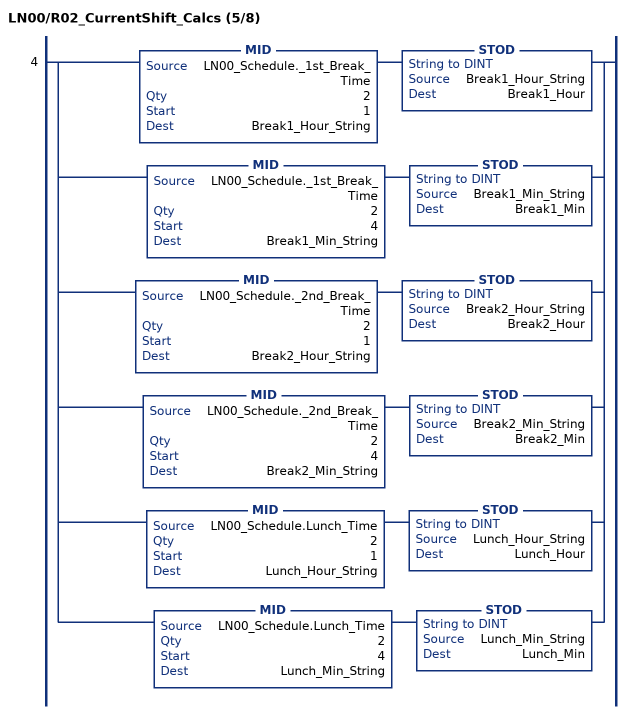
   4: [MID(LN00_Schedule._1st_Break_Time,2,1,Break1_Hour_String) STOD(Break1_Hour_String,Break1_Hour) ,MID(LN00_Schedule._1st_Break_Time,2,4,Break1_Min_String) STOD(Break1_Min_String,Break1_Min) ,MID(LN00_Schedule._2nd_Break_Time,2,1,Break2_Hour_String) STOD(Break2_Hour_String,Break2_Hour) ,MID(LN00_Schedule._2nd_Break_Time,2,4,Break2_Min_String) STOD(Break2_Min_String,Break2_Min) ,MID(LN00_Schedule.Lunch_Time,2,1,Lunch_Hour_String) STOD(Lunch_Hour_String,Lunch_Hour) ,MID(LN00_Schedule.Lunch_Time,2,4,Lunch_Min_String) STOD(Lunch_Min_String,Lunch_Min) ];
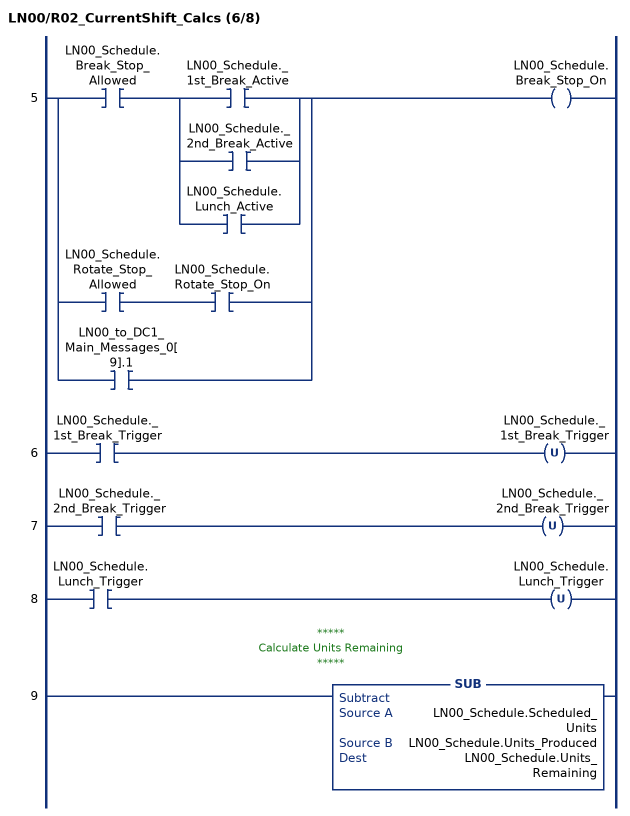
   5: [[XIC(LN00_Schedule.Break_Stop_Allowed) [XIC(LN00_Schedule._1st_Break_Active) ,XIC(LN00_Schedule._2nd_Break_Active) ,XIC(LN00_Schedule.Lunch_Active) ] ,XIC(LN00_Schedule.Rotate_Stop_Allowed) XIC(LN00_Schedule.Rotate_Stop_On) ] ,XIC(LN00_to_DC1_Main_Messages_0[9].1) ]OTE(LN00_Schedule.Break_Stop_On);
   6: XIC(LN00_Schedule._1st_Break_Trigger)OTU(LN00_Schedule._1st_Break_Trigger);
   7: XIC(LN00_Schedule._2nd_Break_Trigger)OTU(LN00_Schedule._2nd_Break_Trigger);
   8: XIC(LN00_Schedule.Lunch_Trigger)OTU(LN00_Schedule.Lunch_Trigger);
   // *****
   // Calculate Units Remaining
   // *****
   9: SUB(LN00_Schedule.Scheduled_Units,LN00_Schedule.Units_Produced,LN00_Schedule.Units_Remaining);
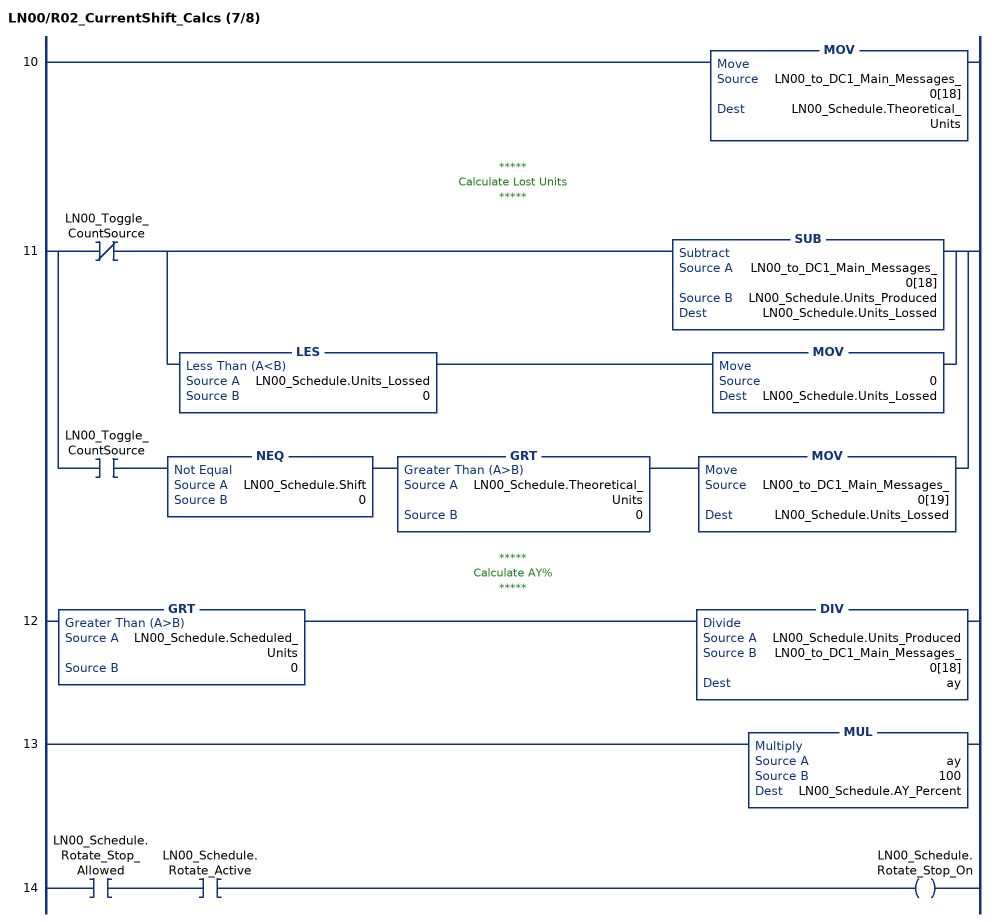
   10: MOV(LN00_to_DC1_Main_Messages_0[18],LN00_Schedule.Theoretical_Units);
   // *****
   // Calculate Lost Units
   // *****
   11: [XIO(LN00_Toggle_CountSource) [SUB(LN00_to_DC1_Main_Messages_0[18],LN00_Schedule.Units_Produced,LN00_Schedule.Units_Lossed) ,LES(LN00_Schedule.Units_Lossed,0) MOV(0,LN00_Schedule.Units_Lossed) ] ,XIC(LN00_Toggle_CountSource) NEQ(LN00_Schedule.Shift,0) GRT(LN00_Schedule.Theoretical_Units,0) MOV(LN00_to_DC1_Main_Messages_0[19],LN00_Schedule.Units_Lossed) ];
   // *****
   // Calculate AY%
   // *****
   12: GRT(LN00_Schedule.Scheduled_Units,0)DIV(LN00_Schedule.Units_Produced,LN00_to_DC1_Main_Messages_0[18],ay);
   13: MUL(ay,100,LN00_Schedule.AY_Percent);
   14: XIC(LN00_Schedule.Rotate_Stop_Allowed)XIC(LN00_Schedule.Rotate_Active)OTE(LN00_Schedule.Rotate_Stop_On);
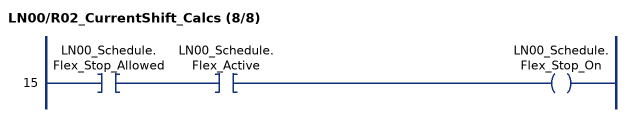
   15: XIC(LN00_Schedule.Flex_Stop_Allowed)XIC(LN00_Schedule.Flex_Active)OTE(LN00_Schedule.Flex_Stop_On);
END_ROUTINE
